{attribute 'qualified_only'}
VAR_GLOBAL
	nLifeSignal				: WORD;
END_VAR

(* stored: Version 1.1.0.1, ProductVersion 3.1.4024.11
   GVL GVL_Python: Id {c57cc303-4ed4-41b6-99b8-c0dafa713aeb} *)
